Universal Robots PolyScope program: measure.urp

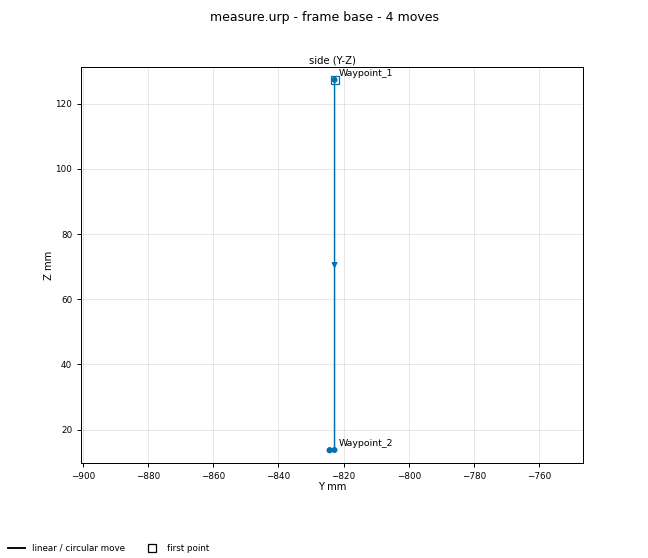
[picture p0: tool path of measure.urp in frame base, 4 of 4 moves have a stored position in this frame; points joined in program order, loops and branches not executed]
Program measure (installation=default directory=/programs/usbdisk/brazo_final/measure createdIn=5.13.0 lastSavedIn=5.13.0 robotSerialNumber=20205500280)
Calibrated DH parameters: a=[0.000126, -0.227628, -0.392536, 0.000072, 0.000053, 0]; d=[0.16267, 78.773992, -78.210517, -0.430145, 0.099656, 0.099678]; alpha=[1.568545, -0.004566, 0.00572, 1.569931, -1.57104, 0]; deltaTheta=[0, -1.006608, 7.298003, -0.008206, 0.000004, 0]
InitVariablesNode
Robot Program (runOnlyOnce=true)
  MoveJ speed 60 deg/s, acceleration 80 deg/s^2 (useActiveTCP=true) feature=Base
    Waypoint Waypoint_1: TCP in base x=-164.038 y=-822.767 z=127.31 mm, rx=-2.1722 ry=2.2503 rz=-0.0153 rad; joints [69.075, -36.777, 30.173, -82.93, -88.935, 71.37] deg; TCP offset x=0 y=0 z=234.35 mm, rx=0 ry=0 rz=-3.1416 rad
    URCap RG6 (RG - On Robot, OnRobot A/S) dataModel(depthCompensate=false, force=120, payload=0.0, width=42, name=RG6(42))
  MoveL speed 250 mm/s, acceleration 1200 mm/s^2 (useActiveTCP=true) feature=Base
    Waypoint Waypoint_2: TCP in base x=-164.011 y=-822.778 z=13.728 mm, rx=-2.1735 ry=2.249 rz=-0.0154 rad; joints [69.051, -36.122, 45.585, -98.999, -88.938, 71.37] deg; TCP offset x=0 y=0 z=234.35 mm, rx=0 ry=0 rz=-3.1416 rad
  Force Frame feature=Base; selection=[0, 1, 0, 0, 0, 0]; wrench=[0, 5, 0, 0, 0, 0]; limitsForce=[0.15, 0.06, 0.15, 1.047198, 1.047198, 1.047198]; limitsMotion=[0.1, 0.1, 0.1, 0.349066, 0.349066, 0.349066]
    Wait Condition expression=ForceYTool<1
    Touch1 := get_actual_tcp_pose()
    lenght1 := (100*Touch1[1])-cal_clavo
  MoveL speed 250 mm/s, acceleration 1200 mm/s^2 (useActiveTCP=true) feature=Base
    Waypoint Waypoint_3: TCP in base x=-164.048 y=-824.276 z=13.657 mm, rx=2.2534 ry=2.1749 rz=0.0219 rad; joints [69.086, -35.834, 45.05, -98.746, -88.941, 251.479] deg; TCP offset x=0 y=0 z=234.35 mm, rx=0 ry=0 rz=-3.1416 rad
    Waypoint Waypoint_4: TCP in base x=-164.034 y=-824.271 z=13.655 mm, rx=2.2513 ry=2.177 rz=0.0219 rad; joints [69.087, -35.834, 45.05, -98.745, -88.942, 251.37] deg; TCP offset x=0 y=0 z=234.35 mm, rx=0 ry=0 rz=-3.1416 rad
  Force Frame feature=Base; selection=[0, 1, 0, 0, 0, 0]; wrench=[0, 5, 0, 0, 0, 0]; limitsForce=[0.15, 0.06, 0.15, 1.047198, 1.047198, 1.047198]; limitsMotion=[0.1, 0.1, 0.1, 0.349066, 0.349066, 0.349066]
    Wait Condition expression=ForceYTool>1
    Touch2 := get_actual_tcp_pose()
    length2 := (100*Touch1[1])-cal_clavo
Thread Thread_1 (runOnlyOnce=false)
  ToolForce := get_tcp_force()
  ForceYTool := ToolForce[1]
  Wait Sleep waitTime=0.01
